	      ELSE // Unsupported character
	        #tempCodepoint := #REPLACEMENT_CHAR;
	        #tempPos += 1;
	        #tempStatus := #WARN_UNSUPPORTED_CHAR;
	      END_IF;

	      // Concatenate decoded characters
	      #tempString := CONCAT(IN1 := #tempString, IN2 := DWORD_TO_WCHAR(#tempCodepoint));

	    UNTIL ((#count <> 0 AND LEN(#tempString) >= #count) OR #tempPos > #tempUpperBound) END_REPEAT;
	  END_IF;
	END_REGION

	REGION OUTPUTS
	  // Write application specific temp values to outputs
	  IF #tempStatus.%X15 = TRUE THEN // An error occured
	    #decodedString := WString#'';
	  ELSE // Successful or with warning
	    #decodedString := #tempString;
	  END_IF;

	  // Write status
	  ENO := #tempStatus.%X15;
	  #LGF_DecodeUtf8 := #tempStatus;
	END_REGION

END_FUNCTION

FUNCTION "LGF_TimeToString" : String
{ S7_Optimized_Access := 'TRUE' }
AUTHOR : Siemens_Digital_Industry
FAMILY : LGF
NAME : LGF_TimeToString
   VAR_INPUT
      timeValue : Time;
   END_VAR

   VAR_OUTPUT
      stringDay : String;
      stringHour : String;
      stringMinute : String;
      stringSecond : String;
      stringMilliSecond : String;
   END_VAR

   VAR_TEMP
      tempTimeResult : String;
      tempTimeMilliseconds : DInt;
      tempDays : DInt;
      tempHours : DInt;
      tempMinutes : DInt;
      tempSecond : DInt;
      tempMillisecond : DInt;
   END_VAR

   VAR CONSTANT
      MS_PER_DAY : DInt := 86400000;
      MS_PER_HOUR : DInt := 3600000;
      MS_PER_MINUTE : DInt := 60000;
      MS_PER_SECOND : DInt := 1000;
      NUMBER_OF_CHAR_TO_DEL : Int := 1;
      FIRST_POSITION : Int := 1;
      NO_REMAINDER : Int := 0;
   END_VAR


BEGIN
	REGION BLOCK INFO HEADER
	  //===============================================================================
	  // SIEMENS AG / (c)Copyright 2017
	  //-------------------------------------------------------------------------------
	  // Title:            LGF_TimeToString
	  // Comment/Function: This function converts a time value to a string
	  //                   When more than one time unit is specified, the value must not exceed 24 days, 23 hours, 59 minutes, 59 seconds or 999 milliseconds.
	  //                   Output format is the folowing := '10D20H30M20S630MS', just existing parts would be added to the string
	  // Library/Family:   LGF(Library General Functions)
	  // Author:           Siemens Digital Industry Support
	  // Tested with:      S7-PLCSIM Advanced V2.0 SP1
	  // Engineering:      TIA Portal V14 SP1 Upd 5
	  // Restrictions:     ENO mechanism is not used, no error handling
	  // Requirements:     PLC (S7-1200 / S7-1500)
	  //-------------------------------------------------------------------------------
	  // Change log table:
	  // Version  | Date       | Expert in charge       | Changes applied
	  //----------|------------|------------------------|------------------------------
	  // 01.00.00 | 03.07.2018 | Siemens Industry Online Support
	  //                         First released version
	  // 01.00.01 | 17.08.2018 | Siemens Industry Online Support
	  //                         Upgrade: TIA V15 Update 2
	  // 01.00.02 | 23.11.2018 | Siemens Industry Online Support
	  //                         Upgrade: TIA V15.1
	  // 01.00.03 | 02.07.2019 | Simatic Systems Support
	  //                         Standard header and block parameters update, status parameter added
	  // 01.00.05 | 09.07.2019 | Simatic Systems Support
	  //                         Further improvements minimization and commends added
	  // 01.00.06 | 30.07.2019 | Simatic Systems Support
	  //                         Add ENO handling
	  // 03.00.00 | 23.04.2020 | Simatic Systems Support | Set version to V3.0.0
	  //                         Harmonize the version of the whole library
	  // 03.00.01 | 23.02.2021 | Simatic Systems Support
	  //                         Insert documentation
	  //===============================================================================
	END_REGION Block info header

	REGION INITIALISATION
	  #tempTimeResult := '';
	END_REGION

	REGION CONVERT
	  // convert from time to millisecond
	  #tempTimeMilliseconds := TIME_TO_DINT(#timeValue);

	  // calculate the days and remaining hours
	  #tempDays := #tempTimeMilliseconds / #MS_PER_DAY;
	  #tempTimeMilliseconds := #tempTimeMilliseconds MOD #MS_PER_DAY;

	  // calculate the hours and remaining minutes
	  #tempHours := #tempTimeMilliseconds / #MS_PER_HOUR;
	  #tempTimeMilliseconds := #tempTimeMilliseconds MOD #MS_PER_HOUR;

	  // calculate the minutes and remaining seconds
	  #tempMinutes := #tempTimeMilliseconds / #MS_PER_MINUTE;
	  #tempTimeMilliseconds := #tempTimeMilliseconds MOD #MS_PER_MINUTE;

	  // calculate the seconds and remaining milliseconds
	  #tempSecond := #tempTimeMilliseconds / #MS_PER_SECOND;
	  #tempMillisecond := #tempTimeMilliseconds MOD #MS_PER_SECOND;

	  // check if value is greater then zero and add to result string without leading "+"
	  IF (#tempMillisecond > #NO_REMAINDER) THEN
	    #stringMilliSecond := DELETE(IN := DINT_TO_STRING(#tempMillisecond), L := #NUMBER_OF_CHAR_TO_DEL, P := #FIRST_POSITION);
	    #tempTimeResult := CONCAT(IN1 := #stringMilliSecond, IN2 := 'MS');
	  END_IF;

	  // check if value is greater then zero and add to result string without leading "+"
	  IF (#tempSecond > #NO_REMAINDER) THEN
	    #stringSecond := DELETE(IN := DINT_TO_STRING(#tempSecond), L := #NUMBER_OF_CHAR_TO_DEL, P := #FIRST_POSITION);
	    #tempTimeResult := CONCAT(IN1 := #stringSecond, IN2 := 'S', IN3 := #tempTimeResult);
	  END_IF;

	  // check if value is greater then zero and add to result string without leading "+"
	  IF (#tempMinutes > #NO_REMAINDER) THEN
	    #stringMinute := DELETE(IN := DINT_TO_STRING(#tempMinutes), L := #NUMBER_OF_CHAR_TO_DEL, P := #FIRST_POSITION);
	    #tempTimeResult := CONCAT(IN1 := #stringMinute, IN2 := 'M', IN3 := #tempTimeResult);
	  END_IF;

	  // check if value is greater then zero and add to result string without leading "+"
	  IF (#tempHours > #NO_REMAINDER) THEN
	    #stringHour := DELETE(IN := DINT_TO_STRING(#tempHours), L := #NUMBER_OF_CHAR_TO_DEL, P := #FIRST_POSITION);
	    #tempTimeResult := CONCAT(IN1 := #stringHour, IN2 := 'H', IN3 := #tempTimeResult);
	  END_IF;

	  // check if value is greater then zero and add to result string without leading "+"
	  IF (#tempDays > #NO_REMAINDER) THEN
	    #stringDay := DELETE(IN := DINT_TO_STRING(#tempDays), L := #NUMBER_OF_CHAR_TO_DEL, P := #FIRST_POSITION);
	    #tempTimeResult := CONCAT(IN1 := #stringDay, IN2 := 'D', IN3 := #tempTimeResult);
	  END_IF;
	END_REGION

	REGION OUTPUTS
	  #LGF_TimeToString := #tempTimeResult;
	  //ENO mechanism is not used - forced to true.
	  ENO := TRUE;
	END_REGION

END_FUNCTION

FUNCTION "LGF_UnixTimeToDTL" : DTL
{ S7_Optimized_Access := 'TRUE' }
AUTHOR : Siemens_Digital_Industry
FAMILY : LGF
NAME : LGF_UnixTimeToDTL
   VAR_INPUT
      timeUnix : DInt;
   END_VAR

   VAR_OUTPUT
      error : Bool;
      status : Word;
   END_VAR

   VAR_TEMP
      tempDate : DInt;
      tempTime : DInt;
      tempDTL {InstructionName := 'DTL'; LibVersion := '1.0'} : DTL;
   END_VAR

   VAR CONSTANT
      DELTA_1970_1990 : DInt := 631_152_000;
      SEC_PER_DAY : DInt := 86400;
      SEC_PER_HOUR : DInt := 3600;
      SEC_PER_MINUTE : DInt := 60;
      STATUS_NO_ERRROR : Word := 16#0000;
      ERR_TIME_BEFORE_1990 : Word := 16#8000;
      WARN_CONVERSION_LIMIT : Word := 16#6001;
      CONVERSION_LIMIT {InstructionName := 'DTL'; LibVersion := '1.0'} : DTL := DTL#1990-01-01-00:00:00;
   END_VAR


BEGIN
	REGION BLOCK INFO HEADER
	  //===============================================================================
	  // SIEMENS AG / (c)Copyright 2017
	  //-------------------------------------------------------------------------------
	  // Title:            LGF_UnixTimeToDTL
	  // Comment/Function: This function converts a Unix time of data type DInt to a date and time of data type DTL.
	  //                   The timestamp is calculated in UTC. This means that the time zone is not taken into account.
	  //                   Only times after 01/01/1990 are permitted.
	  // Library/Family:   LGF (Library General Functions)
	  // Author:           Siemens Digital Industry Support
	  // Tested with:      S7-PLCSIM Advanced V2.0 SP1
	  // Engineering:      TIA Portal V15
	  // Restrictions:     ENO mechanism is not used, Error handling done by error and status
	  // Requirements:     PLC (S7-1200 / S7-1500)
	  //-------------------------------------------------------------------------------
	  // Change log table:
	  // Version  | Date       | Expert in charge       | Changes applied
	  //----------|------------|------------------------|------------------------------
	  // 01.00.00 | 16.10.2018 | Siemens Industry Online Support
	  //                         First released version
	  // 01.00.01 | 18.06.2019 | Simatic Systems Support
	  //                         Standard header and block parameters update, status parameter added
	  // 01.00.02 | 10.07.2019 | Simatic Systems Support
	  //                         Commends added and code intention adjusted
	  //                         Add ENO handling
	  // 03.00.00 | 23.04.2020 | Simatic Systems Support | Set version to V3.0.0
	  //                         Harmonize the version of the whole library
	  // 03.00.01 | 23.02.2021 | Simatic Systems Support
	  //                         Insert documentation
	  //=============================================================================
	END_REGION Block info header

	REGION CONVERT
	  // Check if timeUnix less than 01.01.1990
	  IF (#timeUnix < #DELTA_1970_1990) THEN
	    #LGF_UnixTimeToDTL := #CONVERSION_LIMIT;
	    #error := TRUE;
	    #status := #ERR_TIME_BEFORE_1990;
	    RETURN;

	    // Check if timeUnix is exactly on lower limitation of 01.01.1990
	  ELSIF (#timeUnix = #DELTA_1970_1990) THEN
	    #LGF_UnixTimeToDTL := #CONVERSION_LIMIT;
	    #error := FALSE;
	    #status := #WARN_CONVERSION_LIMIT;
	    RETURN;
	  END_IF;

	  // Convert date
	  #tempDate := (#timeUnix - #DELTA_1970_1990) / #SEC_PER_DAY;
	  #tempDTL := DATE_TO_DTL(DINT_TO_DATE(#tempDate));

	  // Convert time
	  #tempTime := #timeUnix - #DELTA_1970_1990 - (#tempDate * #SEC_PER_DAY);
	  #tempDTL.HOUR := DINT_TO_USINT(#tempTime / #SEC_PER_HOUR);
	  #tempDTL.MINUTE := DINT_TO_USINT(#tempTime MOD #SEC_PER_HOUR / #SEC_PER_MINUTE);
	  #tempDTL.SECOND := DINT_TO_USINT(#tempTime MOD #SEC_PER_MINUTE);
	END_REGION

	REGION OUTPUTS
	  #LGF_UnixTimeToDTL := #tempDTL;
	  #error := FALSE;
	  #status := #STATUS_NO_ERRROR;
	  //ENO mechanism is not used - forced to true.
	  ENO := TRUE;
	END_REGION

END_FUNCTION

